// TIA Portal V16 export
// export: Created 2024-12-03T15:41:41.0474891Z, ExportSetting WithDefaults, DisplayName Totally Integrated Automation Portal, DisplayVersion V16 Update 6, DisplayName TIA Portal Version Control Interface, DisplayVersion V16 Update 2, DisplayName TIA Portal Openness, DisplayVersion V16 Update 6, DisplayName TIA Portal Teamcenter Gateway, DisplayVersion V16, DisplayName SINAMICS Startdrive Advanced, DisplayVersion V16 Update 5, DisplayName SINAMICS Startdrive G130, G150, S120, S150, SINAMICS MV, S210, DisplayVersion V16 Update 5, DisplayName SINAMICS Startdrive G110M, G120, G120C, G120D, G120P, G115D, DisplayVersion V16 Update 5, DisplayName STEP 7 Professional, DisplayVersion V16 Update 6, DisplayName STEP 7 Safety, DisplayVersion V16, DisplayName WinCC Advanced / Unified PC, DisplayVersion V16 Update 6
FUNCTION_BLOCK "HmiButton"   // FB8, SCL
{ S7_Optimized_Access := 'FALSE' }
VERSION : 0.1
// stored: AutoNumber true, IsIECCheckEnabled false, SetENOAutomatically false, UDAEnableTagReadback false
   VAR_INPUT
      I_Enable : Bool;
      I_Flash : Bool;
      I_Type : Int;   // 0 = push button | 1 = toggle button
   END_VAR
   VAR_IN_OUT
      ButtonStatus : "HMIButton_UDT";
   END_VAR
   VAR
      S_smartbool { S7_SetPoint := 'True'} : "SmartBool";
   END_VAR
   VAR_TEMP
      T_Signal : Bool;
   END_VAR
BEGIN
   #T_Signal := #I_Enable AND #ButtonStatus.SignalFromHMI;

   REGION Determine color

       IF NOT #I_Enable OR (#I_Flash AND "Clock_0.5Hz" AND #ButtonStatus.colorNumber = 0) THEN
           #ButtonStatus.colorNumber := -1;
       ELSE
           #ButtonStatus.colorNumber := 0;
       END_IF;

   END_REGION

   REGION "SmartBool"
       #S_smartbool(I_Sensor := #T_Signal,
                    O_data=>#ButtonStatus.state);

   END_REGION

   IF #I_Type = 0 AND #ButtonStatus.SignalFromHMI AND NOT #ButtonStatus.state.LE THEN
       #ButtonStatus.SignalFromHMI := 0;
   END_IF;
END_FUNCTION_BLOCK
